TYPE ST_RecStatus ://过程纠偏
STRUCT
    bError             :BOOL;     //纠偏故障
    bRuning           :BOOL;    //纠偏运行中
END_STRUCT
END_TYPE

(* stored: Version 1.1.0.1, ProductVersion 3.1.4024.9
   DUT ST_RecStatus: Id {a749125e-424c-4cf0-9de9-f33839723cf8} *)
